TEXTLIST ServicesConfigTabsTextList
  0 = 'Timing'
   = ''
END_TEXTLIST

(* stored: Version 1.1.0.1, ProductVersion 3.1.4018.5
   TextList ServicesConfigTabsTextList: Id {c351a554-bc80-478b-9bac-049ed32ae017} *)
